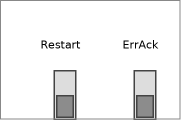
VISUALIZATION Safety  // 181x120
    DipSwitch (40,70 50x50), variable: MAIN.Restart, behaviour: TOGGLE, style: Switch-DipSwitch-Gray
    Label (20,30 81x30), "Restart"
    DipSwitch (120,70 50x50), variable: MAIN.ErrAck, behaviour: TOGGLE, style: Switch-DipSwitch-Gray
    Label (100,30 81x30), "ErrAck"
END_VISUALIZATION

(* stored: Version 1.1.0.1, ProductVersion 3.1.4026.8
   Visu Safety: Id {2c72abb1-52b7-4434-8d69-25eedaf9331f} *)
